// TIA Portal V19 export
FUNCTION "CIPTank" : Void   // FC44, STL
TITLE = CIP ASEPTIC TANK
{ S7_Optimized_Access := 'TRUE' }
NAME : CIPTANK
VERSION : 0.0
// Setpoints to Cip forward changed to real from integer
// stored: AutoNumber false
BEGIN

NETWORK
TITLE = CIP ASEPTIC TANK
      AN    "S0 CIP TANK";
      R     "S1 CIP TANK";
      R     "S2 CIP TANK";
      R     "S3 CIP TANK";
      R     "S4 CIP TANK";
      R     "S5 CIP TANK";
      R     "S6 CIP TANK";
      R     "S7 CIP TANK";
      R     "S8 CIP TANK";
      R     "S9 CIP TANK";
      R     "S10 CIP TANK";
      R     "S11 CIP TANK";
      R     "S12 CIP TANK";
      R     "S13 CIP TANK";
      R     "S14 CIP TANK";
      R     "S15 CIP TANK";
      R     "S16 CIP TANK";
      R     "S17 CIP TANK";
      R     "S18 CIP TANK";
      R     "S19 CIP TANK";
      R     "S20 CIP TANK";
      BEC;
      A     "S1 CIP TANK";
      JC    M001;
      R     "MY0545";
      R     "MY0148";
      R     "MY0103";
      R     "MY0104";
      R     "MY0101";
      R     "MY0112";
      R     "MY0113";
      R     "MY0116";
      R     "MY0117";
      S     "MY0118";
      R     "MY0147";
      R     "MY0143";
      S     "MY0111";
      R     "MY0137";
      R     "MY0136";
      R     "MY0108";
      R     "MY0124";
//    R     "MM01.30"
      R     "CT_LYE_OK";
      R     "CT_ACID_OK";
      R     "MY0109";
//    L     "Setpoints".PT0167SpCIP     //"DB SETPOINTS".PT0167SpCIP
      L     "Setpoints".PT0167SpCIPLow;
      T     "STP_PT0167/IP0149_50".PT0167SpSTP;
//    L     "Setpoints".PT0167SpCIP     //"DB SETPOINTS".PT0167SpCIP
      L     "Setpoints".PT0167SpCIPLow;
      L     0.1;
      -R;
      T     "Setpoints".StartCipMinPressure;  //"DB SETPOINTS".StartCipMinPressure
      S     "AutoPT0167/IP0149";
      S     "LowCIPPressure";
      R     "AcidCipPressure";

//;
      R     "M_Barrier_Sterile";
      R     "M_Product_Route";
      R     "M_Product_Available";
      R     "MY0901";
      R     "MY0906";
      S     "MY0907";
      S     "MY0912";
//;
      A     "Y0907S";  //check valve energised
      A     "Y0912S";  //check valve energised
      JCN   M002;

      S     "S1 CIP TANK";
M002: BEU;
M001: NOP   0;

NETWORK
TITLE = 
      A     "S2 CIP TANK";
      JC    c001;

// Wait for measured pressure < max start pressure (min start pressure + 0.2 bar)
// Change because if start cip after production, then too high pressure

      L     "Setpoints".StartCipMinPressure;
      L     0.2;
      +R;
      L     "MeasuredValues".PT0167REAL;
      <R;
      BEC;

      L     "MeasuredValues".PT0167REAL;  // "DB-ANALOG INPUT".PT0167REAL
      L     "Setpoints".StartCipMinPressure;  //"DB SETPOINTS".StartCipMinPressure
      <R;
      BEC;
      S     "MY0113";
      S     "MY0114";
      S     "MY0104";
      S     "MY0115";
      S     "CONTROL CIP TANK";
      S     "S2 CIP TANK";
      BEU;
c001: NOP   0;

NETWORK
TITLE = REGULATOR TT01.72/IP01.57 IN AUTO MODE
// Check balance tank level, feedback correct on V01.13, V01.14, V01.04.
// Load temp set point for pre-rinse and transfer to regulator. Regulator to auto. 
// Open steam supply valve 01.58. Start circulation pump 01.39. Open route to 
// spray 
// ball through V01.03. Start delay open timer V01.12. Step on.
      A     "S3 CIP TANK";
      JC    c002;
      AN    "B01.41";
      BEC;
      AN    "Y0113S";
      BEC;
      AN    "Y0114S";
      BEC;
      AN    "Y0104S";
      BEC;
      L     "Setpoints".TT0172SpPrerinse;
      T     "PID_TT0172/IP0157".TT0172SpDBD;
      S     "AutoTT0172/IP0157";
      S     "MY0158";
      S     "MM0139";
      S     "MY0103";
      S     "TIM18";
      S     "S3 CIP TANK";
      BEU;
c002: NOP   0;

NETWORK
TITLE = Q 8.5; Output modul 1 Channel 5
// Start Pre-rinse timer. Open V01.12. Set V01.08 to pulse. (V01.35 / 36 / 37 & 
// 01.30 not used). Step on.
      A     "S4 CIP TANK";
      JC    c003;
      A     "T 18 DELAY 01.12";
      BEC;
      S     "MY0112";
      S     "TIM27";
      S     "SPIN 01.30 CIP";
      S     "PULSE 01.08 CIP";
      S     "MY0136";
      S     "MY0137";
      R     "MY0135";
      S     "S4 CIP TANK";
      BEU;
c003: NOP   0;

NETWORK
TITLE = Q 8.7; Output modul 1 Channel 7
// If pre-rinse timer has expired, reset V01.014 (route to rec-irculate), set 
// V01.13 ready to pulse, step on.
      A     "S5 CIP TANK";
      JC    c004;
      A     "T 27 WATER 1";
      BEC;
      R     "MY0114";
      S     "PULSE 01.13 CIP";
      S     "S5 CIP TANK";
      BEU;
c004: NOP   0;

NETWORK
TITLE = ProcessAlarm
// Check to see if chemical dosing is already active. Load temp set point for 
// caustic and request caustic dosing. Step on.
      A     "S6 CIP TANK";
      JC    c005;
      A     "R.CIP UNIT OCCUPIED";
      S     "ProcessAndPbAlarms"."A"[43];  //A43_WaitingForCipUnit// waiting for cip unit
      BEC;
      L     "Setpoints".TT0172SpLye;  //"DB SETPOINTS".TT0172SpLye
      T     "PID_TT0172/IP0157".TT0172SpDBD;
      S     "S.T.01.REQUEST LYE";
      S     "S6 CIP TANK";
      BEU;
c005: NOP   0;

NETWORK
TITLE = TANK IS CLEAN
// Comment
      A     "S7 CIP TANK";
      JC    c006;
      AN    "R.CIP UNIT OCCUPIED";
      BEC;
//      S     "TIM28"
      R     "TANK CLEAN";
      S     "S7 CIP TANK";
      BEU;
c006: NOP   0;

NETWORK
TITLE = REQUEST LYE SEND TO UHT FROM TANK 01.00 MPI NET
// Comment  Wait for lye concentration to be OK
      A     "S8 CIP TANK";
      JC    c007;
//    A     "T 28 DOSING LYE"
      AN    "CT_LYE_OK";
      BEC;
      R     "S.T.01.REQUEST LYE";
      R     "CT_LYE_OK";
      R     "LowCIPPressure";
      S     "S8 CIP TANK";
      BEU;
c007: NOP   0;

NETWORK
TITLE = 
// Comment  Wait for return temperature to be OK
      A     "S9 CIP TANK";
      JC    c008;
      L     "MeasuredValues".TT0180REAL;  // "DB-ANALOG INPUT".TT0180MEAS
      L     "Setpoints".MinCipReturTempTT01;  //"DB SETPOINTS".MinCipReturTempTT01
      <R;
      BEC;
      S     "TIM29";
      S     "S9 CIP TANK";
      BEU;
c008: NOP   0;

NETWORK
TITLE = 
// Comment
      A     "S10 CIP TANK";
      JC    c009;
      A     "T 29 LYE CIRCULATION";
      BEC;
      S     "MY0114";
      R     "CONTROL CIP TANK";
      L     25.0;
      T     "PID_TT0172/IP0157".TT0172SpDBD;
//      T     "PID_TT0172/IP0157".TT0172SpPID
      S     "PULSE 01.13 CIP";
      S     "S10 CIP TANK";
      S     "LowCIPPressure";
      R     "AcidCipPressure";
      BEU;
c009: NOP   0;

NETWORK
TITLE = 
// Comment
      A     "S11 CIP TANK";
      JC    c010;
      A     "B01.42";
      BEC;
      S     "CONTROL CIP TANK";
      AN    "LEDAssignment".K4_LIGHT;  //"LIGHT_K4_CIP_LYE"
      S     "TIM30";
      S     "S11 CIP TANK";
      BEC;
      S     "TIM33";
      S     "S18 CIP TANK";
      S     "S17 CIP TANK";
      S     "S16 CIP TANK";
      S     "S15 CIP TANK";
      S     "S14 CIP TANK";
      S     "S13 CIP TANK";
      S     "S12 CIP TANK";
      S     "S11 CIP TANK";
      BEU;
c010: NOP   0;

NETWORK
TITLE = 
// Comment
      A     "S12 CIP TANK";
      JC    c011;
      A     "T 30 WATER 2";
      BEC;
      R     "MY0114";
      S     "PULSE 01.13 CIP";
      S     "S12 CIP TANK";
      S     "AcidCipPressure";
      R     "LowCIPPressure";
      BEU;
c011: NOP   0;

NETWORK
TITLE = A43_WaitingForCipUnit
      A     "S13 CIP TANK";
      JC    c012;
      A     "R.CIP UNIT OCCUPIED";
      S     "ProcessAndPbAlarms"."A"[43];  //A43_WaitingForCipUnit// waiting for cip unit
      BEC;
      L     "Setpoints".PT0167AcidPressure;
      L     0.1;
      +R;
      L     "MeasuredValues".PT0167REAL;
      <R;
      BEC;
      L     "Setpoints".TT0172SpAcid;  //"DB SETPOINTS".TT0172SpAcid
      T     "PID_TT0172/IP0157".TT0172SpDBD;
      S     "S.T.01.REQUEST ACID";
      S     "S13 CIP TANK";
      BEU;
c012: NOP   0;

NETWORK
TITLE = STEP 14 CIP
// Comment
      A     "S14 CIP TANK";
      JC    c013;
      AN    "R.CIP UNIT OCCUPIED";
      BEC;
//    S     "TIM31"
      S     "S14 CIP TANK";
      BEU;
c013: NOP   0;

NETWORK
TITLE = REQUEST ACID SEND TO UHT FROM TANK 01.00 MPI NET
// Comment  Wait for acid concentration to be OK
      A     "S15 CIP TANK";
      JC    c014;
//    A     "T 31 DOSING ACID"
      AN    "CT_ACID_OK";
      BEC;
      R     "S.T.01.REQUEST ACID";
      R     "CT_ACID_OK";
      S     "S15 CIP TANK";
      BEU;
c014: NOP   0;

NETWORK
TITLE = 
// Comment
      A     "S16 CIP TANK";
      JC    c015;
      L     "MeasuredValues".TT0180REAL;  // "DB-ANALOG INPUT".TT0180MEAS
      L     "Setpoints".MinCipReturTempTT01;  //"DB SETPOINTS".MinCipReturTempTT01
      <R;
      BEC;
      S     "TIM32";
      S     "LowCIPPressure";
      R     "AcidCipPressure";
      S     "S16 CIP TANK";
      BEU;
c015: NOP   0;

NETWORK
TITLE = Q 8.7; Output modul 1 Channel 7
// Comment
      A     "S17 CIP TANK";
      JC    c016;
      A     "T 32 ACID CIRCULATION";
      BEC;
      S     "MY0114";
      R     "CONTROL CIP TANK";
      S     "PULSE 01.13 CIP";
      L     25.0;
      T     "PID_TT0172/IP0157".TT0172SpDBD;
//      T     "PID_TT0172/IP0157".TT0172SpPID
      S     "S17 CIP TANK";
      BEU;
c016: NOP   0;

NETWORK
TITLE = 
// Comment
      A     "S18 CIP TANK";
      JC    c017;
      A     "B01.42";
      BEC;
      S     "CONTROL CIP TANK";
      S     "TIM33";
      S     "S18 CIP TANK";
      BEU;
c017: NOP   0;

NETWORK
TITLE = CONTROL LEVEL IN CIP TANK
// Comment
      A     "S19 CIP TANK";
      JC    c018;
      A     "T 33 WATER 3";
      BEC;
      R     "CONTROL CIP TANK";
      R     "MM0139";
      R     "MY0158";
      R     "AutoTT0172/IP0157";
      R     "ManTT0172/IP0157";
      R     "MY0103";
      R     "MY0104";
      R     "AutoPT0167/IP0149";
      R     "ManPT0167/IP0149";
      S     "TIM34";
      S     "TANK CLEAN";
      S     "PULSE 01.13 CIP";
      R     "LowCIPPressure";
      R     "AcidCipPressure";
//;
      S     "MY0907";
      S     "MY0912";
      A     "Y0907S";  //check valve energised
      A     "Y0912S";  //check valve energised
      JCN   M003;
//;

      S     "S19 CIP TANK";
M003: BEU;
c018: NOP   0;

NETWORK
TITLE = MAIN FLAG CIP
// Comment
      A     "S20 CIP TANK";
      JC    c019;
      A     "T 34 BLOW OUT CIP";
      BEC;
      R     "S0 CIP TANK";
//;
      R     "MY0907";
      R     "MY0912";
//;
      BEU;
c019: NOP   0;
END_FUNCTION
